FUNCTION_BLOCK Room_State_Fault EXTENDS _Room_State
VAR_INPUT
END_VAR
VAR_OUTPUT
END_VAR
VAR
END_VAR

METHOD PROTECTED OnEntry
_ctx.io.bOpenValves := FALSE;

_ctx.priv.bActive := FALSE;
_ctx.priv.bReady := FALSE;

_ctx.hmi.sStatusText := CONCAT('Fault: ', _ctx.hmi.sErrorText);
_ctx.hmi.nStatusColor := COL.RED.Raw;

_ctx.hmi.bHideReset := FALSE;
END_METHOD

METHOD PROTECTED OnExecute
IF _ctx.hmi.bReset THEN
	_ctx.hmi.bReset := FALSE;
	
	_ctx.state.iMgr.Request(_ctx.state.iIdle);
END_IF
END_METHOD

METHOD PROTECTED OnExit
_ctx.hmi.sErrorText := 'Undefined';
END_METHOD

END_FUNCTION_BLOCK

(* stored: Version 1.1.0.1
   POU Room_State_Fault: Id {a0562641-f5c5-4611-ac4d-a35e1468e2c4}, SpecialFunc None
   Method OnEntry: Id {cbcebeb3-12c0-4102-a8d1-f2f2ae32ad3f}
   Method OnExecute: Id {f6c9b6aa-bf70-4df1-a873-0dcf2557902c}
   Method OnExit: Id {9733460b-de5e-4bd7-ba80-0494bdfd5f66} *)
